Fanuc KAREL source: compact_preamble.KL

PROGRAM KC00040
%NOLOCKGROUP
%ENVIRONMENT IOSETUP
VAR
I:INTEGER;J:INTEGER;K:INTEGER;R:REAL;B:BOOLEAN;S : STRING[80];T : STRING[80];AI : ARRAY[8] OF INTEGER
AB : ARRAY[244] OF BYTE
-- UNRESOLVED DECLARATIONS (source type spelling not recovered)
-- P : TYPE_0x001F (type_u16=0x001F)
-- Q : TYPE_0x001F (type_u16=0x001F)
BEGIN
GET_PORT_SIM(I,J,B,K)
END KC00040
